(* CODESYS project SM_HOME.library
   Description: Device support for Home Automation board under Raspberry Pi
   Version: 1.1.0.0
   Title: Raspberry I2C HOME AUTOMATION
   Author: Sequent Microsystems
   DocFormat: reStructuredText
   LanguageModelAttribute: qualified-access-only
   Placeholder: PlaceholderTemplate
   DefaultNamespace: SM_HOME
   Company: Sequent Microsystems

Project tree, tasks and I/O mapping:
  libraries: Raspberry Pi Peripherals, 4.6.0.0 (3S - Smart Software Solutions GmbH); IoStandard, 3.5.17.0 (System); Standard, 3.5.18.0 (System)
  global variables GVL
  function block SM_HOME [ST]: AfterReadInputs, BeforeWriteOutputs
  Library Information/
    function GetLibVersionNumber [ST]
    function GetLibVersion [ST]
    function IsLibReleased [ST]
  Project Information/
    function GetCompany [ST]
    function GetTitle [ST]
    function GetVersion [ST]
    function GetTextProperty [ST]
    function GetTextProperty2 [ST]
    function GetNumberProperty [ST]
    function GetBooleanProperty [ST]
    function GetVersionProperty [ST]
*)

// GVL
//{attribute 'qualified_only'}
VAR_GLOBAL CONSTANT
	RELAY_VAL_ADD: USINT := 16#00;
	RELAY_SET_ADD: USINT := 16#01;
	RELAY_CLR_ADD: USINT := 16#02;
	OPTO_VAL_ADD: USINT := 16#03;
	
	U0_10_OUT_VAL1_ADD: USINT := 16#28;
	U0_3_IN_VAL1_ADD: USINT := 16#18;
	OD_PWM1_ADD:USINT:= 16#30;
	TEMPERATURE_ADD: USINT := 16#3E;
	OWB_DEV_COUNT_ADD: USINT := 16#D3;
	OWB_TEMP1_ADD: USINT := 16#DE;
	
END_VAR

// SM_HOME
FUNCTION_BLOCK SM_HOME EXTENDS i2c
VAR_INPUT
	relayState: ARRAY[0..7] OF BOOL;
	out0_10Volt: ARRAY[0..3] OF REAL;
	outOdPwm:ARRAY[0..3] OF REAL;
END_VAR
VAR_OUTPUT
	inOpto: ARRAY[0..7] OF BOOL;
	in0_3Volt: ARRAY[0..7] OF REAL;
	inOWBTemp: ARRAY[0..7] OF REAL;
	inOWBSensors: USINT;
	boardTemperature: REAL;
END_VAR
VAR
	timer: TON := (IN:=TRUE);
	relayStateRaw: USINT;
	out0_10VoltRaw: ARRAY[0..3] OF UINT;
	outOdPwmRaw: ARRAY[0..3] OF UINT;
	readOWBCount: USINT;
END_VAR
VAR_TEMP	
	i, usi: USINT;
	buff: ARRAY[0..20] OF USINT;	
END_VAR

SUPER^();

CASE _iState OF
0:
	IF usiAddress < 16#28 OR  usiAddress > 16#30 THEN
		usiAddress := 16#28;
	END_IF
	//usiAddress := 16#31 + StackLevel;
	IF SUPER^.init() THEN
		_iState := 5;
	END_IF	
5:	
	Timer.pt := T#20MS;
	buff[1] := 0;
	buff[2] := 0;
	FOR i:=0 TO 3 DO
		buff[0] := U0_10_OUT_VAL1_ADD + i* 2;
		write(ADR(buff), 3);
		out0_10VoltRaw[i] := 0;
	END_FOR
	
	// init all relay off
	
	relayStateRaw := 0;
	write8(RELAY_VAL_ADD, 0);
	readOWBCount:=0;
	
	_iState := 10;
END_CASE

METHOD AfterReadInputs:INT
VAR
	Buffer : ARRAY[0..3] OF BYTE;
	ch: USINT;
	address: USINT;
	value: REAL;
	len: DINT;	
	opto: USINT;
END_VAR
SUPER^.AfterReadInputs();

IF _iState = 10 THEN
	timer(IN:=TRUE);
	IF timer.Q THEN	
		opto := read8(OPTO_VAL_ADD);  
		FOR len:=0 TO 7 DO
			inOpto[len] := USINT_TO_BOOL(SHL(2#00000001, len) AND opto);
		END_FOR
	
		boardTemperature := read8(TEMPERATURE_ADD);
		IF readOWBCount < 20 THEN
			readOWBCount := readOWBCount + 1;	
		ELSE
			readOWBCount := 0;
			inOWBSensors := read8(OWB_DEV_COUNT_ADD);	
			IF inOWBSensors > 0 THEN
				FOR ch:=0 TO inOWBSensors - 1 DO
					address:= OWB_TEMP1_ADD + 2*ch;
					len := readregister(address, ADR(Buffer), 2);		
					IF len = 2 THEN
						value := BYTE_TO_REAL(Buffer[0]) + BYTE_TO_REAL(Buffer[1]) * 256;
						inOWBTemp[ch]:=value/100;
					END_IF
				END_FOR
			END_IF
		END_IF
	
		
		FOR ch:=0 TO 7 DO
			address:= U0_3_IN_VAL1_ADD + 2*ch;
			len := readregister(address, ADR(Buffer), 2);		
			IF len = 2 THEN
				value := BYTE_TO_REAL(Buffer[0]) + BYTE_TO_REAL(Buffer[1]) * 256;
				in0_3Volt[ch]:=value/1000;
			END_IF
		END_FOR
		
		timer(IN:=FALSE);
	END_IF
END_IF
END_METHOD

METHOD BeforeWriteOutputs:INT
VAR
	i: USINT;
	cnt: USINT;
	inVal:UINT;
	inSVal:USINT;
	buff: ARRAY[0..2] OF USINT;
	wStat: BOOL;
END_VAR
SUPER^.BeforeWriteOutputs();

IF _iState = 10 THEN

	
	FOR i:=0 TO 3 DO
		IF out0_10Volt[i] < 0 THEN
			out0_10Volt[i] := 0;
		END_IF
		IF out0_10Volt[i] > 10 THEN
			out0_10Volt[i] := 10;
		END_IF
		inVal := REAL_TO_UINT(out0_10Volt[i] * 1000);
		IF out0_10VoltRaw[i] <> inVal THEN
			buff[0] := U0_10_OUT_VAL1_ADD + 2*i;
			buff[2] := UINT_TO_USINT(inVal / 256);
			buff[1] := UINT_TO_USINT(inVal - (inVal / 256));
			cnt := DINT_TO_USINT(write(ADR(buff), 3));
			IF cnt = 3 THEN
				out0_10VoltRaw[i] := inVal;
			END_IF	
		END_IF
	END_FOR  
	
	FOR i:=0 TO 3 DO
		IF outOdPwm[i] < 0 THEN
			outOdPwm[i] := 0;
		END_IF
		IF outOdPwm[i] > 100 THEN
			outOdPwm[i] := 100;
		END_IF
		inVal := REAL_TO_UINT(outOdPwm[i] * 100);
		IF outOdPwmRaw[i] <> inVal THEN
			buff[0] := OD_PWM1_ADD + 2*i;
			buff[2] := UINT_TO_USINT(inVal / 256);
			buff[1] := UINT_TO_USINT(inVal - (inVal / 256));
			cnt := DINT_TO_USINT(write(ADR(buff), 3));
			IF cnt = 3 THEN
				outOdPwmRaw[i] := inVal;
			END_IF	
		END_IF
	END_FOR  
	
	inSVal:= 0;
	FOR i:= 0 TO 7 DO
		inSVal:= inSVal + SHL(BOOL_TO_USINT(relayState[i]), i);
	END_FOR
	IF relayStateRaw <> inSVal THEN
		IF write8(RELAY_VAL_ADD, inSVal) THEN
			relayStateRaw:=inSVal;
		END_IF
	END_IF		
END_IF
END_METHOD

END_FUNCTION_BLOCK

// Library Information/GetLibVersionNumber
// This function has been automatically generated from the project information.
FUNCTION GetLibVersionNumber : DWORD
VAR_INPUT
	
END_VAR

GetLibVersionNumber := 16842752;

END_FUNCTION

// Project Information/GetCompany
// This function has been automatically generated from the project information.
{attribute 'signature_flag' := '1073741824'}
{attribute 'register_in_runtime'}
FUNCTION GetCompany : WSTRING
VAR_INPUT
	
END_VAR

GetCompany := "Sequent Microsystems";

END_FUNCTION

// Project Information/GetTitle
// This function has been automatically generated from the project information.
{attribute 'signature_flag' := '1073741824'}
{attribute 'register_in_runtime'}
FUNCTION GetTitle : WSTRING
VAR_INPUT
	
END_VAR

GetTitle := "Raspberry I2C HOME AUTOMATION";

END_FUNCTION

// Library Information/GetLibVersion
// This function has been automatically generated from the project information.
FUNCTION GetLibVersion : VERSION
VAR_INPUT
	
END_VAR

GetLibVersion.uiMajor := 1;
GetLibVersion.uiMinor := 1;
GetLibVersion.uiServicePack := 0;
GetLibVersion.uiPatch := 0;

END_FUNCTION

// Library Information/IsLibReleased
// This function has been automatically generated from the project information.
FUNCTION IsLibReleased : BOOL
VAR_INPUT
	
END_VAR

IsLibReleased := FALSE;

END_FUNCTION

// Project Information/GetVersion
// This function has been automatically generated from the project information.
{attribute 'signature_flag' := '1073741824'}
{attribute 'register_in_runtime'}
FUNCTION GetVersion : VERSION
VAR_INPUT
	
END_VAR

GetVersion.uiMajor := 1;
GetVersion.uiMinor := 1;
GetVersion.uiServicePack := 0;
GetVersion.uiPatch := 0;

END_FUNCTION

// Project Information/GetTextProperty
// This function has been automatically generated from the project information.
{attribute 'signature_flag' := '1073741824'}
{attribute 'register_in_runtime'}
FUNCTION GetTextProperty : WSTRING
VAR_INPUT
	stKey: WSTRING;
END_VAR

IF stKey = "Author" THEN
	GetTextProperty := "Sequent Microsystems";
ELSIF stKey = "Company" THEN
	GetTextProperty := "Sequent Microsystems";
ELSIF stKey = "DefaultNamespace" THEN
	GetTextProperty := "SM_HOME";
ELSIF stKey = "Description" THEN
	GetTextProperty := "Device support for Home Automation board under Raspberry Pi";
ELSIF stKey = "DocFormat" THEN
	GetTextProperty := "reStructuredText";
ELSIF stKey = "LanguageModelAttribute" THEN
	GetTextProperty := "qualified-access-only";
ELSIF stKey = "Placeholder" THEN
	GetTextProperty := "PlaceholderTemplate";
ELSIF stKey = "Project" THEN
	GetTextProperty := "SM_HOME";
ELSIF stKey = "Title" THEN
	GetTextProperty := "Raspberry I2C HOME AUTOMATION";
ELSE
	GetTextProperty := "";
END_IF

END_FUNCTION

// Project Information/GetTextProperty2
// This function has been automatically generated from the project information.
{attribute 'signature_flag' := '1073741824'}
{attribute 'register_in_runtime'}
FUNCTION GetTextProperty2 : POINTER TO WSTRING
VAR_INPUT
	stKey: WSTRING;
END_VAR

IF stKey = "Author" THEN
	GetTextProperty2 := ADR("Sequent Microsystems");
ELSIF stKey = "Company" THEN
	GetTextProperty2 := ADR("Sequent Microsystems");
ELSIF stKey = "DefaultNamespace" THEN
	GetTextProperty2 := ADR("SM_HOME");
ELSIF stKey = "Description" THEN
	GetTextProperty2 := ADR("Device support for Home Automation board under Raspberry Pi");
ELSIF stKey = "DocFormat" THEN
	GetTextProperty2 := ADR("reStructuredText");
ELSIF stKey = "LanguageModelAttribute" THEN
	GetTextProperty2 := ADR("qualified-access-only");
ELSIF stKey = "Placeholder" THEN
	GetTextProperty2 := ADR("PlaceholderTemplate");
ELSIF stKey = "Project" THEN
	GetTextProperty2 := ADR("SM_HOME");
ELSIF stKey = "Title" THEN
	GetTextProperty2 := ADR("Raspberry I2C HOME AUTOMATION");
ELSE
	GetTextProperty2 := ADR("");
END_IF

END_FUNCTION

// Project Information/GetNumberProperty
// This function has been automatically generated from the project information.
{attribute 'signature_flag' := '1073741824'}
{attribute 'register_in_runtime'}
FUNCTION GetNumberProperty : DINT
VAR_INPUT
	stKey: WSTRING;
END_VAR

GetNumberProperty := 0;

END_FUNCTION

// Project Information/GetBooleanProperty
// This function has been automatically generated from the project information.
{attribute 'signature_flag' := '1073741824'}
{attribute 'register_in_runtime'}
FUNCTION GetBooleanProperty : BOOL
VAR_INPUT
	stKey: WSTRING;
END_VAR

IF stKey = "IsEndUserLibrary" THEN
	GetBooleanProperty := FALSE;
ELSIF stKey = "Released" THEN
	GetBooleanProperty := FALSE;
ELSE
	GetBooleanProperty := FALSE;
END_IF

END_FUNCTION

// Project Information/GetVersionProperty
// This function has been automatically generated from the project information.
{attribute 'signature_flag' := '1073741824'}
{attribute 'register_in_runtime'}
FUNCTION GetVersionProperty : VERSION
VAR_INPUT
	stKey: WSTRING;
END_VAR

IF stKey = "Version" THEN
	GetVersionProperty.uiMajor := 1;
	GetVersionProperty.uiMinor := 1;
	GetVersionProperty.uiServicePack := 0;
	GetVersionProperty.uiPatch := 0;
ELSE
	GetVersionProperty.uiMajor := 0;
	GetVersionProperty.uiMinor := 0;
	GetVersionProperty.uiServicePack := 0;
	GetVersionProperty.uiPatch := 0;
END_IF

END_FUNCTION
